// TwinCAT 3 PLC project TeamsPlc
// Title: TeamsApp
// Company: TcOpen
// ProjectVersion: 0.0.0.0
// ProgramVersion: 3.1.4023.0
// libraries:
//   Tc2_Standard, * (Beckhoff Automation GmbH)
//   Tc2_System, * (Beckhoff Automation GmbH)
//   Tc3_Module, * (Beckhoff Automation GmbH)
//   TcoCore, 0.4.2.453 (Vortex.Library)
// project tree:
//   / PlcTask.TcTTO
//   POUs/ MAIN.TcPOU, TeamsApp.TcPOU
// real-time tasks:
//   TASK PlcTask: cycle T#10ms, priority 20, ADS port 350

CONFIGURATION TeamsPlc
    RESOURCE PLC ON TwinCAT3
        TASK PlcTask(INTERVAL := T#10ms, PRIORITY := 20);
        PROGRAM MAIN WITH PlcTask : MAIN;
    END_RESOURCE
END_CONFIGURATION

// ---- POUs/MAIN.TcPOU
PROGRAM MAIN
VAR
	App : TeamsApp;
END_VAR

App.Run();

END_PROGRAM

// ---- POUs/TeamsApp.TcPOU
FUNCTION_BLOCK TeamsApp EXTENDS TcoContext
VAR
	StartTheMachine : TcoCore.TcoTask(THIS^);
	StopTheMachine : TcoCore.TcoTask(THIS^);
	
	IsMachineRunning : BOOL;
	MessageFromPlc : STRING;
END_VAR

(*~
	<docu>
		<summary>
			Main method of the TcoContext. This is the entry point of any control logic that belongs to this context. 
			The call of this method is ensured by calling the <c>InstanceName.Run()</c> method, and it must not be called explicitly.
			This method is abstract, and it must be overridden in derived block.
		</summary>
	</docu>
~*)
METHOD PROTECTED  Main
IF StartTheMachine.Execute() THEN
    IF IsMachineRunning THEN
        MessageFromPlc := 'The machine is already running!';
    ELSE
        MessageFromPlc := '';
    END_IF

    IsMachineRunning := TRUE;
    StartTheMachine.DoneWhen(IsMachineRunning);
END_IF

IF StopTheMachine.Execute() THEN
    IF NOT IsMachineRunning THEN
        MessageFromPlc := 'The machine is already off!';
    ELSE
        MessageFromPlc := '';
    END_IF

    IsMachineRunning := FALSE;
    StopTheMachine.DoneWhen(NOT IsMachineRunning);
END_IF
END_METHOD

END_FUNCTION_BLOCK
